// TIA Portal V20 export
// export: Created 2026-04-11T06:02:30.6044529Z, ExportSetting WithDefaults, DisplayName Totally Integrated Automation Portal, DisplayVersion V20, DisplayName TIA Portal Openness, DisplayVersion V20, DisplayName TIA Portal Version Control Interface, DisplayVersion V20, DisplayName STEP 7 Professional, DisplayVersion V20, DisplayName STEP 7 Safety, DisplayVersion V20, DisplayName WinCC Basic/Comfort/Advanced, DisplayVersion V20, DisplayName WinCC Unified, DisplayVersion V20
TYPE "udtHMI_Brabender_Status"
// stored: IsFailsafeCompliant false
   STRUCT
      bInterLockedStopped { ExternalWritable := 'False'} : Bool;   // WORD 10 Bit 0: Feeder Interlocked and stopped
      bInterLockedStarted { ExternalWritable := 'False'} : Bool;   // WORD 16 Bit 1: Feeder Interlocked and started
      bControlDiffPos { ExternalWritable := 'False'} : Bool;   // WORD 16 Bit 2: Control difference +
      bControlDiffNeg { ExternalWritable := 'False'} : Bool;   // WORD 16 Bit 3: Control Difference -
      bStarted { ExternalWritable := 'False'} : Bool;   // WORD 16 Bit 4: Feeder started
      bAlarm { ExternalWritable := 'False'} : Bool;   // WORD 16 Bit 5: Alarm
      bRefilAutoTareBypass { ExternalWritable := 'False'} : Bool;   // WORD 16 Bit 6: Refill Auto-tare Bypass
      bAlarmReport { ExternalWritable := 'False'} : Bool;   // WORD 16 Bit 7: Alarm Report
      bBatchEndDropOut { ExternalWritable := 'False'} : Bool;   // WORD 17 Bit 2: Batch end Drop-out
      bBTEnabled { ExternalWritable := 'False'} : Bool;   // WORD 17 Bit 3: Operation BT field bus locked(0); enabled(1)
      bStatusOP1 { ExternalWritable := 'False'} : Bool;   // WORD 17 Bit 4: Status OP1 0 = Interlocked(off); 1 = enabled(on)
      bAntiVibration { ExternalWritable := 'False'} : Bool;   // WORD 17 Bit 6: Anti-Vibration
      bStabilizationTime { ExternalWritable := 'False'} : Bool;   // WORD 17 Bit 7: Stabilization Time
   END_STRUCT;
END_TYPE
